// TIA Portal project "S7-1200" (V18)

(* hardware
DEVICE "S7-1200 station_1"  S7-1200 Station
   slot 0: "Rack_0"  S7-1200 Rack  Rack  V1.0
   slot 1: "PLC_2"  CPU 1212C AC/DC/Rly  6ES7 212-1BE40-0XB0  V4.6
*)

// ===== PLC "PLC_2"  CPU 1212C AC/DC/Rly =====

VAR_GLOBAL   // PLC tag table "Default tag table_1"
   "Tag_1" AT %M0.0 : Bool;
   "Tag_2" AT %Q0.3 : Bool;
   "Tag_3" AT %Q0.4 : Bool;
   "Tag_4" AT %M0.2 : Bool;
   "Tag_5" AT %M0.1 : Bool;
   "Tag_6" AT %Q0.5 : Bool;
   "Tag_7" AT %Q0.6 : Bool;
   "Tag_8" AT %Q0.7 : Bool;
   "Tag_9" AT %Q1.0 : Bool;
END_VAR

VAR_GLOBAL CONSTANT   // PLC tag table "Default tag table_1"
   "None(1)" : Pip := 65535;
   "Automatic update(1)" : Pip := 0;
   "PIP 1(1)" : Pip := 1;
   "PIP 2(1)" : Pip := 2;
   "PIP 3(1)" : Pip := 3;
   "PIP 4(1)" : Pip := 4;
   "PIP 5" : Pip := 5;
   "PIP 6" : Pip := 6;
   "PIP 7" : Pip := 7;
   "PIP 8" : Pip := 8;
   "PIP 9" : Pip := 9;
   "PIP 10" : Pip := 10;
   "PIP 11" : Pip := 11;
   "PIP 12" : Pip := 12;
   "PIP 13" : Pip := 13;
   "PIP 14" : Pip := 14;
   "PIP 15" : Pip := 15;
   "PIP 16" : Pip := 16;
   "PIP 17" : Pip := 17;
   "PIP 18" : Pip := 18;
   "PIP 19" : Pip := 19;
   "PIP 20" : Pip := 20;
   "PIP 21" : Pip := 21;
   "PIP 22" : Pip := 22;
   "PIP 23" : Pip := 23;
   "PIP 24" : Pip := 24;
   "PIP 25" : Pip := 25;
   "PIP 26" : Pip := 26;
   "PIP 27" : Pip := 27;
   "PIP 28" : Pip := 28;
   "PIP 29" : Pip := 29;
   "PIP 30" : Pip := 30;
   "PIP 31" : Pip := 31;
   "PIP OB Servo(1)" : Pip := 32768;
   "Local~MC(1)" : Hw_SubModule := 51;
   "Local~Common(1)" : Hw_SubModule := 50;
   "Local~Device(1)" : Hw_Device := 32;
   "Local~Configuration(1)" : Hw_SubModule := 33;
   "Local~Display" : Hw_SubModule := 54;
   "Local~Exec(1)" : Hw_SubModule := 52;
   "Local(1)" : Hw_SubModule := 49;
   "Local~PROFINET_interface_1(1)" : Hw_Interface := 64;
   "Local~PROFINET_interface_1~Port_1(1)" : Hw_Interface := 65;
   "Local~PROFINET_interface_1~Port_2" : Hw_Interface := 66;
   "Local~Virtual_communication_interface" : Hw_Interface := 135;
   "Local~License_Manager" : Hw_SubModule := 42;
   "OB_Main(1)" : OB_PCYCLE := 1;
END_VAR

ORGANIZATION_BLOCK "Main"   // OB1, LAD, ProgramCycle
TITLE = "Main Program Sweep (Cycle)"
{ S7_Optimized_Access := 'TRUE' }
VERSION : 0.1
   VAR_INPUT
      Initial_Call : Bool;   // Initial call of this OB
      Remanence : Bool;   // =True, if remanent data are available
   END_VAR
BEGIN

REGION Network 1
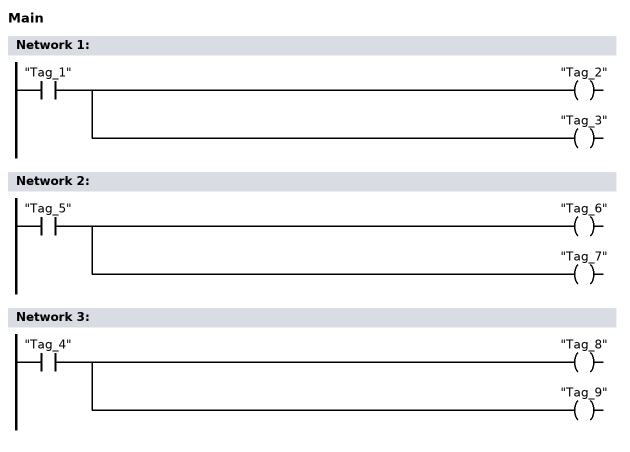
   RUNG wire#powerrail
      Contact( "Tag_1" )
      wire#w1
      Coil( "Tag_2" )
   END_RUNG
   RUNG wire#w1
      Coil( "Tag_3" )
   END_RUNG
   // the same network as SCL:
   "Tag_2" := "Tag_1";
   "Tag_3" := "Tag_1";
END_REGION

REGION Network 2
   RUNG wire#powerrail
      Contact( "Tag_5" )
      wire#w1
      Coil( "Tag_6" )
   END_RUNG
   RUNG wire#w1
      Coil( "Tag_7" )
   END_RUNG
   // the same network as SCL:
   "Tag_6" := "Tag_5";
   "Tag_7" := "Tag_5";
END_REGION

REGION Network 3
   RUNG wire#powerrail
      Contact( "Tag_4" )
      wire#w1
      Coil( "Tag_8" )
   END_RUNG
   RUNG wire#w1
      Coil( "Tag_9" )
   END_RUNG
   // the same network as SCL:
   "Tag_8" := "Tag_4";
   "Tag_9" := "Tag_4";
END_REGION
END_ORGANIZATION_BLOCK